(* Schneider Machine Expert - Basic project Exercise-7 - Set and Reset LEDs, file version 2.9.0.0 *)
(* ProjectInformations: Name=New project *)

HARDWARE
  Cpu 0: TM221CE24R
  EthernetConfiguration: NetworkName=M221, IpAllocationMode=FixedAddress, IpAddress=0.0.0.0, SubnetMask=0.0.0.0
  SerialLineConfiguration: Baud=Baud19200, Parity=ParityEven, DataBits=DataBits8, StopBits=StopBits1, PhysicalMedium=PhysicalMediumRs485, SlaveId=1, Addressing=SlaveAddressing
  MastTask: UsePeriodScanMode=false, PeriodScan=100
  FastTask: Period=255
  CpuBehavior: StartingMode=StartAsPreviousState, AutoSaveRamOnEeprom=true, WatchdogPeriod=250

SYMBOLS  (address, symbol, comment, settings)
  %I0.0     SWITCH_1
  %I0.1     SWITCH_2
  %I0.2     RESET_SWITCH
  %Q0.0     LED_1
  %Q0.1     LED_2
  %Q0.2     LED_3
  %Q0.3     LED_4

POU New POU
  (* SectionNumber=1 *)

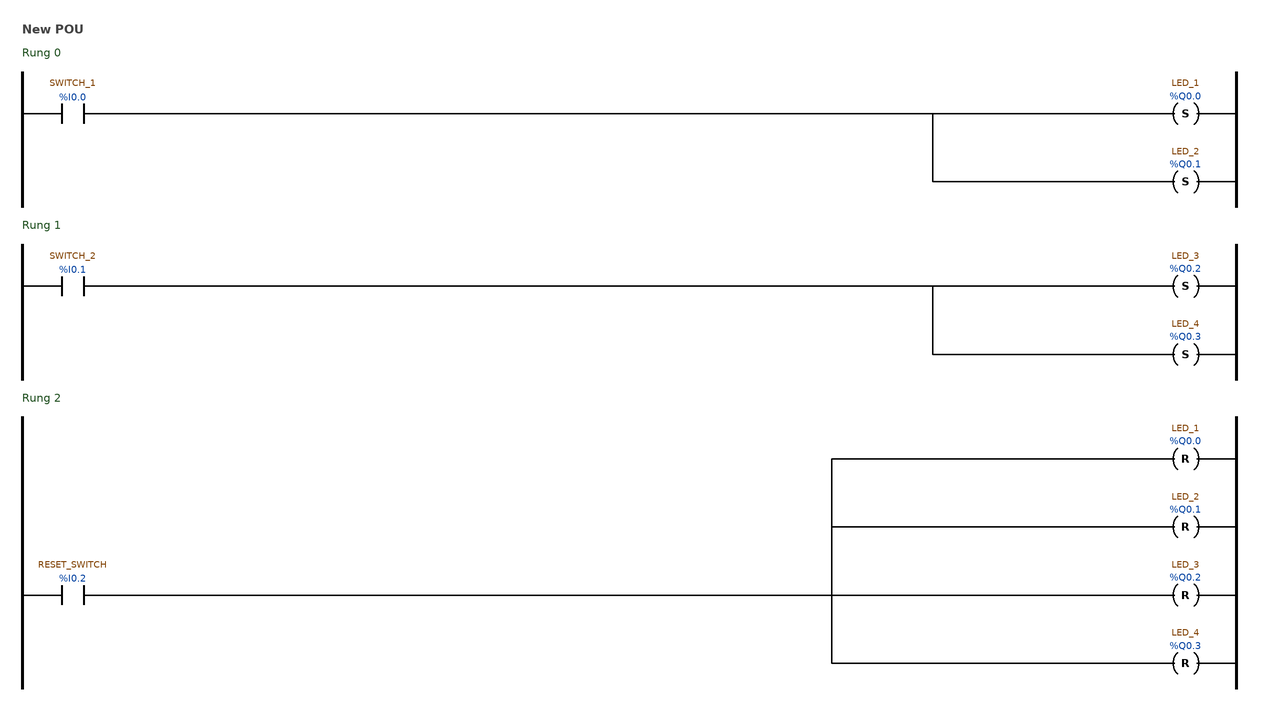

// Rung 0
  LD %I0.0                (* SWITCH_1 *)
  S %Q0.0                 (* LED_1 *)
  S %Q0.1                 (* LED_2 *)
  // as ST:
  //   IF SWITCH_1 THEN LED_1 := TRUE; END_IF;
  //   IF SWITCH_1 THEN LED_2 := TRUE; END_IF;

// Rung 1
  LD %I0.1                (* SWITCH_2 *)
  S %Q0.2                 (* LED_3 *)
  S %Q0.3                 (* LED_4 *)
  // as ST:
  //   IF SWITCH_2 THEN LED_3 := TRUE; END_IF;
  //   IF SWITCH_2 THEN LED_4 := TRUE; END_IF;

// Rung 2
  LD %I0.2                (* RESET_SWITCH *)
  R %Q0.0                 (* LED_1 *)
  R %Q0.1                 (* LED_2 *)
  R %Q0.2                 (* LED_3 *)
  R %Q0.3                 (* LED_4 *)
  // as ST:
  //   IF RESET_SWITCH THEN LED_1 := FALSE; END_IF;
  //   IF RESET_SWITCH THEN LED_2 := FALSE; END_IF;
  //   IF RESET_SWITCH THEN LED_3 := FALSE; END_IF;
  //   IF RESET_SWITCH THEN LED_4 := FALSE; END_IF;
